// TIA Portal project "Conveyor_Box" (V18)

(* hardware
DEVICE "S7-1200 station_1"  S7-1200 Station
   slot 0: "Rack_0"  S7-1200 Rack  Rack  V1.0
   slot 1: "192.168.20.60"  CPU 1212C AC/DC/Rly  6ES7 212-1BE40-0XB0  V4.6
   slot 2: "DI 8/DQ 8x24VDC_1"  SM 1223 DI8/DQ8 x 24VDC  6ES7 223-1BH30-0XB0  V1.0
*)

// ===== PLC "192.168.20.60"  CPU 1212C AC/DC/Rly =====

VAR_GLOBAL   // PLC tag table "In"
   "Inputs" AT %I0.0 : "In";   // Digital Inputs
   "Inputs_DM" AT %I8.0 : "In_DM";
END_VAR

VAR_GLOBAL   // PLC tag table "Out"
   "Outputs" AT %Q0.0 : "Out";   // Digital Outputs
   "Outputs_DM" AT %Q2.0 : "Out_DM";
END_VAR

TYPE "In"
   STRUCT
      Emergency_Stop : Bool;   // Emergency stop push
      PB_Start : Bool;   // Pushbutton start normally open
      PB_Stop : Bool;   // Pushbutton stop normally close
      Sensor_Cylinder_Box_A : Bool;   // Photoelectric sensor final conveyor
      Sensor_Cylinder_Box_B : Bool;   // Photoelectric sensor medium conveyor
      Cylinder_Sensor_Back_A : Bool;   // Back sensor cylinder A
      Cylinder_Sensor_Front_A : Bool;   // Front sensor cylinder A
      Cylinder_Sensor_Back_B : Bool;   // Back sensor cylinder B
   END_STRUCT;
END_TYPE

TYPE "Out"
   STRUCT
      Cylinder_A : Bool;   // Cylinder stamp A
      Cylinder_B : Bool;   // Cylinder stamp B
      Cylinder_C : Bool;   // Cylinder push box
      "Conveyor_A-0" : Bool;   // Conveyor one first part
      "Conveyor_A-1" : Bool;   // Conveyor one second part
      Conveyor_B : Bool;   // Conveyor two
   END_STRUCT;
END_TYPE

TYPE "In_DM"
   STRUCT
      Cylinder_Sensor_Front_B : Bool;   // Front sensor cylinder B
      Sensor_Box_Conveyor_B : Bool;   // Sensor box start conveyor B
      Sensor_H_Box : Bool;   // Sensor detect height
      Final_Sensor_Conveyor : Bool;   // Final sensor conveyor A-1
      Cylinder_Sensor_Back_C : Bool;   // Back sensor cylinder C
      Cylinder_Sensor_Front_C : Bool;   // Front sensor cylinder C
   END_STRUCT;
END_TYPE

TYPE "Out_DM"
   STRUCT
      Run_Pilot : Bool;   // Run process green light indicator
      Stop_Pilot : Bool;   // Stop process red light indicator
   END_STRUCT;
END_TYPE

DATA_BLOCK "Global_Var"   // DB1
{ S7_Optimized_Access := 'TRUE' }
VERSION : 0.1
   VAR
      In : "In";   // Physical inputs plc
      In_DM : "In_DM";   // Physical inputs digital module
      Out : "Out";   // Physical outputs plc
      Out_DM : "Out_DM";   // Physical outputs digital module
      Start_Stop : Bool;
   END_VAR
BEGIN
END_DATA_BLOCK

FUNCTION "Start_stop_process" : Void   // FC1, LAD
TITLE = Start stop process
{ S7_Optimized_Access := 'TRUE' }
AUTHOR : Stiven Perez Mora
VERSION : 0.1
// conditions to start or stop all process
   VAR_INPUT
      Pb_Start : Bool;
      Emergency_Stop : Bool;
      Pb_Stop : Bool;
   END_VAR
   VAR_IN_OUT
      Run_Pilot : Bool;
      Stop_Pilot : Bool;
   END_VAR
BEGIN

REGION Network 1: start
   // conditions to start all process
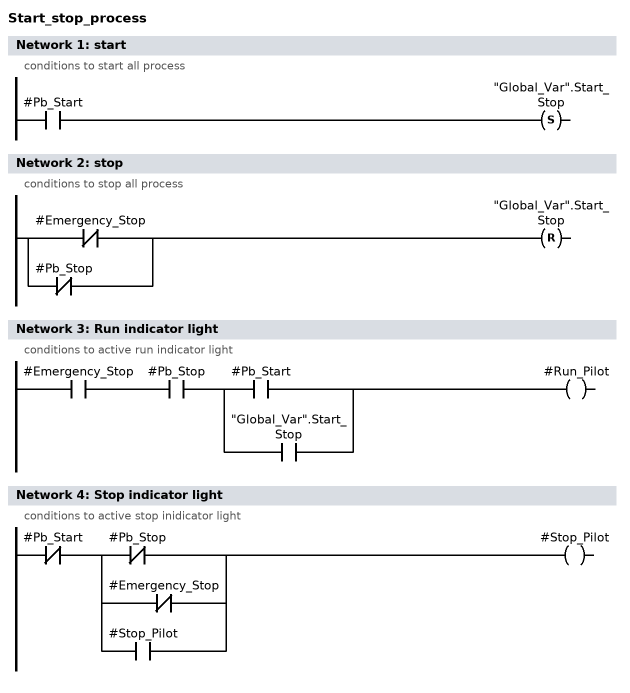
   RUNG wire#powerrail
      Contact( #Pb_Start )
      S_Coil( "Global_Var".Start_Stop )
   END_RUNG
   // the same network as SCL:
   IF #Pb_Start THEN "Global_Var".Start_Stop := TRUE; END_IF;
END_REGION

REGION Network 2: stop
   // conditions to stop all process
   RUNG wire#powerrail
      I_Contact( #Emergency_Stop )
      wire#w1
      R_Coil( "Global_Var".Start_Stop )
   END_RUNG
   RUNG wire#powerrail
      I_Contact( #Pb_Stop )
   END_RUNG wire#w1
   // the same network as SCL:
   IF NOT #Emergency_Stop OR NOT #Pb_Stop THEN "Global_Var".Start_Stop := FALSE; END_IF;
END_REGION

REGION Network 3: Run indicator light
   // conditions to active run indicator light
   RUNG wire#powerrail
      Contact( #Emergency_Stop )
      Contact( #Pb_Stop )
      wire#w1
      Contact( #Pb_Start )
      wire#w2
      Coil( #Run_Pilot )
   END_RUNG
   RUNG wire#w1
      Contact( "Global_Var".Start_Stop )
   END_RUNG wire#w2
   // the same network as SCL:
   #Run_Pilot := #Emergency_Stop AND #Pb_Stop AND (#Pb_Start OR "Global_Var".Start_Stop);
END_REGION

REGION Network 4: Stop indicator light
   // conditions to active stop inidicator light
   RUNG wire#powerrail
      I_Contact( #Pb_Start )
      wire#w1
      I_Contact( #Pb_Stop )
      wire#w2
      Coil( #Stop_Pilot )
   END_RUNG
   RUNG wire#w1
      I_Contact( #Emergency_Stop )
   END_RUNG wire#w2
   RUNG wire#w1
      Contact( #Stop_Pilot )
   END_RUNG wire#w2
   // the same network as SCL:
   #Stop_Pilot := NOT #Pb_Start AND (NOT #Pb_Stop OR NOT #Emergency_Stop OR #Stop_Pilot);
END_REGION
END_FUNCTION

ORGANIZATION_BLOCK "Main"   // OB1, LAD, ProgramCycle
TITLE = "Main Program Sweep (Cycle)"
{ S7_Optimized_Access := 'TRUE' }
VERSION : 0.1
   VAR_INPUT
      Initial_Call : Bool;   // Initial call of this OB
      Remanence : Bool;   // =True, if remanent data are available
   END_VAR
BEGIN
END_ORGANIZATION_BLOCK